{attribute 'qualified_only'}
VAR_GLOBAL CONSTANT
	MaxStateCount : INT := 5;
	MaxTransitionCount : INT := 20;
END_VAR

(* stored: Version 1.1.0.1
   GVL ProgramConstants: Id {c578cc40-d567-45be-b86a-0847989f2715} *)
